(****************************************************************************************)
(*							Beckhoff Automation Poland									*)
(*									F_1stByteW	v1.0									*)
(*									15.02.2010											*)
(*		Funkcja wyciagajaca mniej znaczacy BYTE ze zmiennej typu WORD					*)
(*							 wyjscie typu WORD											*)
(*______________________________________________________________________________________*)
FUNCTION F_1stByteW : WORD
VAR_INPUT
	wIn:	WORD;
END_VAR

F_1stByteW := wIn AND 16#FF;

END_FUNCTION

(* stored: Version 1.1.0.1, ProductVersion 3.1.4020.3
   POU F_1stByteW: Id {2548d8cf-d639-4a8e-b341-312f9939f085}, SpecialFunc None *)
